% RSLogix 500 project Generator-Start-Stop-Control-I-O-Mapping-&-Emulator-Troubleshooting.RSS, saved by version 8.30.00.16 %
PROJECT "GENSTART"    % processor: Bul.1763 MicroLogix 1100 Series B %

PROGRAM FILES
  LAD 2 "MAIN"  3 rungs
  LAD 3 "DIGITAL IO"  7 rungs
  LAD 4 "CONTROLS"  4 rungs

DATA FILES
  O0 OUTPUT  6 elements
  I1 INPUT  6 elements
  S2 STATUS  66 elements
  B3 BINARY  1 elements
  T4 TIMER  1 elements
  C5 COUNTER  1 elements
  R6 CONTROL  1 elements
  N7 INTEGER  1 elements
  F8 FLOAT  1 elements

LADDER 2 "MAIN"
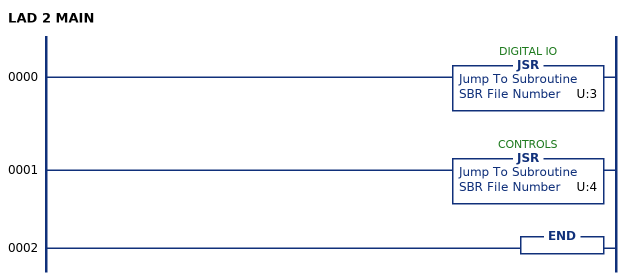
% Rung: 0 %
SOR JSR U:3 EOR
%   U:3  "DIGITAL IO" %
% Rung: 1 %
SOR JSR U:4 EOR
%   U:4  "CONTROLS" %
% Rung: 2 %
SOR END EOR

LADDER 3 "DIGITAL IO"
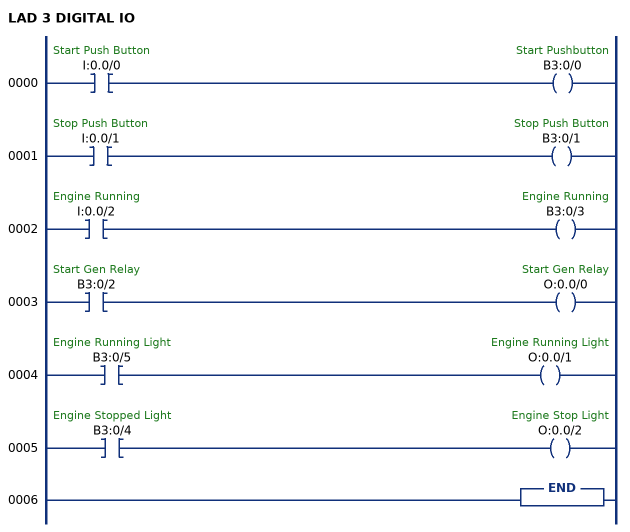
% Rung: 0 %
SOR XIC I:0.0/0 OTE B3:0/0 EOR
%   I:0.0/0  "Start Push Button" %
%   B3:0/0  "Start Pushbutton" %
% Rung: 1 %
SOR XIC I:0.0/1 OTE B3:0/1 EOR
%   I:0.0/1  "Stop Push Button" %
%   B3:0/1  "Stop Push Button" %
% Rung: 2 %
SOR XIC I:0.0/2 OTE B3:0/3 EOR
%   I:0.0/2  "Engine Running" %
%   B3:0/3  "Engine Running" %
% Rung: 3 %
SOR XIC B3:0/2 OTE O:0.0/0 EOR
%   B3:0/2  "Start Gen Relay" %
%   O:0.0/0  "Start Gen Relay" %
% Rung: 4 %
SOR XIC B3:0/5 OTE O:0.0/1 EOR
%   B3:0/5  "Engine Running Light" %
%   O:0.0/1  "Engine Running Light" %
% Rung: 5 %
SOR XIC B3:0/4 OTE O:0.0/2 EOR
%   B3:0/4  "Engine Stopped Light" %
%   O:0.0/2  "Engine Stop Light" %
% Rung: 6 %
SOR END EOR

LADDER 4 "CONTROLS"
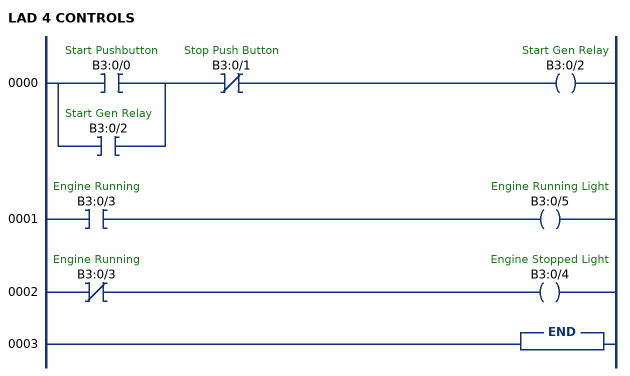
% Rung: 0 %
SOR BST XIC B3:0/0 NXB XIC B3:0/2 BND XIO B3:0/1 OTE B3:0/2 EOR
%   B3:0/0  "Start Pushbutton" %
%   B3:0/2  "Start Gen Relay" %
%   B3:0/1  "Stop Push Button" %
% Rung: 1 %
SOR XIC B3:0/3 OTE B3:0/5 EOR
%   B3:0/3  "Engine Running" %
%   B3:0/5  "Engine Running Light" %
% Rung: 2 %
SOR XIO B3:0/3 OTE B3:0/4 EOR
%   B3:0/3  "Engine Running" %
%   B3:0/4  "Engine Stopped Light" %
% Rung: 3 %
SOR END EOR

OTHER DOCUMENTED ADDRESSES
  I:0.0/3  "Engine Stopped Light"
  I:0.0/4  "Engine Start Light"
  U:2  "MAIN"

DATA TABLE (non-zero values as saved)
DATA B3
% B3:0 % 0X002D
